{attribute 'qualified_only'}
VAR_GLOBAL
	AX_StructModbusTCP 	AT %MW112 	: ARRAY[1..10000] OF WORD;
END_VAR

(* stored: Version 1.1.0.1, ProductVersion 3.1.4024.9
   GVL GVL_DataBaseStructures: Id {de53c85b-c590-4350-88b0-e296727641ab} *)
